(* IEC 61131-3 sources: horner-cscape-mcp/fixtures/st_programs, 6 files *)

(* ---- analog_scaling_program.st ---- *)
(* ============================================================================
 * Title:       PROGRAM AnalogScalingApp
 * Description: Multichannel Process Analog Signal Conditioner with Bounds Checking.
 * Features:
 *   - 4-Channel transmitter linear scaling to engineering units
 *   - Independent out-of-bounds detection: Wire-break and short-circuit faults
 *   - Safe value substitution during hardware transducer failure
 *   - Process alarms for high and low limit excursions
 *   - Master diagnostic health word encoding for SCADA / HMI telemetry
 * Language:    IEC 61131-3 Structured Text (Pure ST)
 * ============================================================================ *)

PROGRAM AnalogScalingApp
VAR_INPUT
    RawCh1 : REAL := 16000.0;             (* Raw ADC Channel 1: Pressure transmitter *)
    RawCh2 : REAL := 18500.0;             (* Raw ADC Channel 2: Temperature transmitter *)
    RawCh3 : REAL := 12000.0;             (* Raw ADC Channel 3: Flow rate transmitter *)
    RawCh4 : REAL := 22000.0;             (* Raw ADC Channel 4: Tank level transmitter *)
    ResetFaults : BOOL := FALSE;          (* Push button to clear sensor fault latches *)
END_VAR

VAR_OUTPUT
    Press_PSIG : REAL := 0.0;             (* Scaled pressure: 0.0 to 150.0 PSIG *)
    Temp_DegC : REAL := 0.0;              (* Scaled temperature: -20.0 to 250.0 Deg C *)
    Flow_GPM : REAL := 0.0;               (* Scaled flow rate: 0.0 to 500.0 GPM *)
    Level_Pct : REAL := 0.0;              (* Scaled vessel level: 0.0 to 100.0 % *)
    Ch1_Fault : BOOL := FALSE;            (* Channel 1 wire break or short circuit *)
    Ch2_Fault : BOOL := FALSE;            (* Channel 2 wire break or short circuit *)
    Ch3_Fault : BOOL := FALSE;            (* Channel 3 wire break or short circuit *)
    Ch4_Fault : BOOL := FALSE;            (* Channel 4 wire break or short circuit *)
    HealthStatusWord : WORD := 16#FFFF;   (* 16-bit status mask (Bit 0-3 = Channel OK) *)
    HighPressureAlarm : BOOL := FALSE;    (* Pressure above 135.0 PSIG warning *)
    HighLevelAlarm : BOOL := FALSE;       (* Level above 90.0 % overflow warning *)
END_VAR

VAR
    RawMinVal : REAL := 3200.0;           (* Raw count corresponding to 4.0 mA *)
    RawMaxVal : REAL := 32000.0;          (* Raw count corresponding to 20.0 mA *)
    BreakThreshold : REAL := 2500.0;      (* Underflow threshold declaring open circuit *)
    ShortThreshold : REAL := 32500.0;     (* Overflow threshold declaring short circuit *)
    SpanCh1 : REAL := 150.0;              (* Range span: Channel 1 *)
    SpanCh2 : REAL := 270.0;              (* Range span: Channel 2 (-20 to 250) *)
    SpanCh3 : REAL := 500.0;              (* Range span: Channel 3 *)
    SpanCh4 : REAL := 100.0;              (* Range span: Channel 4 *)
    RawSpan : REAL := 28800.0;            (* RawSpan = 32000 - 3200 *)
END_VAR

(* 1. Fault Clear *)
IF ResetFaults THEN
    Ch1_Fault := FALSE;
    Ch2_Fault := FALSE;
    Ch3_Fault := FALSE;
    Ch4_Fault := FALSE;
END_IF;

(* 2. Channel 1: Steam Header Pressure (0.0 to 150.0 PSIG) *)
IF RawCh1 < BreakThreshold OR RawCh1 > ShortThreshold THEN
    Ch1_Fault := TRUE;
    Press_PSIG := 0.0; (* Fail-safe pressure reading *)
ELSE
    Press_PSIG := ((RawCh1 - RawMinVal) / RawSpan) * SpanCh1;
    Press_PSIG := LIMIT(0.0, Press_PSIG, 150.0);
END_IF;

(* 3. Channel 2: Reactor Fluid Temperature (-20.0 to 250.0 Deg C) *)
IF RawCh2 < BreakThreshold OR RawCh2 > ShortThreshold THEN
    Ch2_Fault := TRUE;
    Temp_DegC := 25.0; (* Fail-safe ambient default *)
ELSE
    Temp_DegC := -20.0 + (((RawCh2 - RawMinVal) / RawSpan) * SpanCh2);
    Temp_DegC := LIMIT(-20.0, Temp_DegC, 250.0);
END_IF;

(* 4. Channel 3: Feed Flow Rate (0.0 to 500.0 GPM) *)
IF RawCh3 < BreakThreshold OR RawCh3 > ShortThreshold THEN
    Ch3_Fault := TRUE;
    Flow_GPM := 0.0; (* Fail-safe zero flow *)
ELSE
    Flow_GPM := ((RawCh3 - RawMinVal) / RawSpan) * SpanCh3;
    Flow_GPM := LIMIT(0.0, Flow_GPM, 500.0);
END_IF;

(* 5. Channel 4: Bulk Storage Tank Level (0.0 to 100.0 %) *)
IF RawCh4 < BreakThreshold OR RawCh4 > ShortThreshold THEN
    Ch4_Fault := TRUE;
    Level_Pct := 0.0; (* Fail-safe empty level *)
ELSE
    Level_Pct := ((RawCh4 - RawMinVal) / RawSpan) * SpanCh4;
    Level_Pct := LIMIT(0.0, Level_Pct, 100.0);
END_IF;

(* 6. Process Excursion Alarms *)
HighPressureAlarm := Press_PSIG >= 135.0 AND (NOT Ch1_Fault);
HighLevelAlarm := Level_Pct >= 90.0 AND (NOT Ch4_Fault);

(* 7. Health Status Diagnostics Word *)
IF (NOT Ch1_Fault) AND (NOT Ch2_Fault) AND (NOT Ch3_Fault) AND (NOT Ch4_Fault) THEN
    HealthStatusWord := 16#000F; (* All 4 channels healthy *)
ELSE
    HealthStatusWord := 16#0000;
END_IF;

END_PROGRAM

(* ---- batch_reactor_program.st ---- *)
(* ============================================================================
 * Title:       PROGRAM BatchReactorApp
 * Description: Automated Chemical Batch Synthesis Sequential Controller.
 * Features:
 *   - Structured sequential batch phases: Fill, Dose, Heat/Mix, Soak, Cool, Drain
 *   - Recipe parameter integration: Target volume, reagent volume, cook time
 *   - Multi-actuator control: Solvent valve, dosing pump, steam, cooling, agitator
 *   - Reactor overpressure and high-temperature emergency abort interlocks
 * Language:    IEC 61131-3 Structured Text (Pure ST)
 * ============================================================================ *)

PROGRAM BatchReactorApp
VAR_INPUT
    BatchStart : BOOL := FALSE;           (* Operator start batch recipe push button *)
    BatchAbort : BOOL := FALSE;           (* Operator emergency abort push button *)
    EStopHealthy : BOOL := TRUE;          (* Safety circuit permissive *)
    CurrentLevelPct : REAL := 0.0;        (* Vessel liquid level (0.0 to 100.0 %) *)
    CurrentTempC : REAL := 22.0;          (* Vessel liquid temperature (Deg C) *)
    VesselPressBar : REAL := 0.5;         (* Internal vessel pressure (Bar) *)
    ResetAbortPB : BOOL := FALSE;         (* Clear latched abort status *)
    TargetSolventPct : REAL := 65.0;      (* Recipe: Solvent target level (%) *)
    CookTempC : REAL := 85.0;             (* Recipe: Target reaction temperature (Deg C) *)
    CookDurationSec : REAL := 120.0;      (* Recipe: Soak hold duration at cook temperature (s) *)
    CoolTempC : REAL := 35.0;             (* Recipe: Target discharge temperature (Deg C) *)
END_VAR

VAR_OUTPUT
    SolventValve : BOOL := FALSE;         (* Feed valve: Bulk solvent *)
    ReagentPump : BOOL := FALSE;          (* Dosing pump: Catalyst / reagent *)
    AgitatorMotor : BOOL := FALSE;        (* Reaction vessel impeller agitator *)
    SteamValve : BOOL := FALSE;           (* Heating jacket steam admission valve *)
    CoolingValve : BOOL := FALSE;         (* Heating jacket chilled water admission *)
    DischargePump : BOOL := FALSE;        (* Product transfer / emptying pump *)
    BatchPhase : INT := 0;                (* Current recipe phase step code *)
    BatchComplete : BOOL := FALSE;        (* Batch cycle finished flag *)
    PressureAlarm : BOOL := FALSE;        (* Overpressure safety shutdown flag *)
    PhaseTimeSec : REAL := 0.0;           (* Elapsed duration in current phase *)
END_VAR

VAR
    ScanSec : REAL := 0.1;                (* Cyclic scan interval (seconds) *)
    DoseTimer : REAL := 0.0;              (* Reagent dosing duration timer *)
    DoseRequiredSec : REAL := 20.0;       (* Dosing run time required *)
END_VAR

(* 1. Safety Interlocks and Overpressure Protection *)
IF ResetAbortPB THEN
    PressureAlarm := FALSE;
END_IF;

IF VesselPressBar >= 3.5 THEN
    PressureAlarm := TRUE;
END_IF;

IF (NOT EStopHealthy) OR BatchAbort OR PressureAlarm THEN
    BatchPhase := 9; (* Emergency Abort *)
END_IF;

(* 2. Sequential Phase Execution *)
CASE BatchPhase OF

    0: (* PHASE_IDLE: Awaiting Recipe Start *)
        SolventValve := FALSE;
        ReagentPump := FALSE;
        AgitatorMotor := FALSE;
        SteamValve := FALSE;
        CoolingValve := FALSE;
        DischargePump := FALSE;
        PhaseTimeSec := 0.0;
        BatchComplete := FALSE;

        IF BatchStart AND EStopHealthy AND (NOT PressureAlarm) THEN
            BatchPhase := 1;
        END_IF;

    1: (* PHASE_CHARGE_SOLVENT: Fill vessel with bulk solvent *)
        SolventValve := TRUE;
        AgitatorMotor := CurrentLevelPct >= 20.0; (* Start agitator once liquid covers impeller *)
        PhaseTimeSec := PhaseTimeSec + ScanSec;

        IF CurrentLevelPct >= TargetSolventPct THEN
            SolventValve := FALSE;
            DoseTimer := 0.0;
            PhaseTimeSec := 0.0;
            BatchPhase := 2;
        END_IF;

    2: (* PHASE_DOSE_REAGENT: Meter chemical catalyst *)
        ReagentPump := TRUE;
        AgitatorMotor := TRUE;
        DoseTimer := DoseTimer + ScanSec;
        PhaseTimeSec := PhaseTimeSec + ScanSec;

        IF DoseTimer >= DoseRequiredSec THEN
            ReagentPump := FALSE;
            PhaseTimeSec := 0.0;
            BatchPhase := 3;
        END_IF;

    3: (* PHASE_HEAT: Apply steam until target cook temperature is reached *)
        AgitatorMotor := TRUE;
        SteamValve := CurrentTempC < CookTempC;
        CoolingValve := FALSE;
        PhaseTimeSec := PhaseTimeSec + ScanSec;

        IF CurrentTempC >= CookTempC THEN
            PhaseTimeSec := 0.0;
            BatchPhase := 4;
        END_IF;

    4: (* PHASE_SOAK: Hold at reaction temperature for recipe duration *)
        AgitatorMotor := TRUE;
        SteamValve := CurrentTempC < CookTempC;
        CoolingValve := CurrentTempC > (CookTempC + 2.0);
        PhaseTimeSec := PhaseTimeSec + ScanSec;

        IF PhaseTimeSec >= CookDurationSec THEN
            SteamValve := FALSE;
            PhaseTimeSec := 0.0;
            BatchPhase := 5;
        END_IF;

    5: (* PHASE_COOL: Circulate chilled water to quench reaction *)
        AgitatorMotor := TRUE;
        SteamValve := FALSE;
        CoolingValve := TRUE;
        PhaseTimeSec := PhaseTimeSec + ScanSec;

        IF CurrentTempC <= CoolTempC THEN
            CoolingValve := FALSE;
            PhaseTimeSec := 0.0;
            BatchPhase := 6;
        END_IF;

    6: (* PHASE_DISCHARGE: Transfer product out of reactor *)
        AgitatorMotor := CurrentLevelPct >= 15.0;
        DischargePump := TRUE;
        PhaseTimeSec := PhaseTimeSec + ScanSec;

        IF CurrentLevelPct <= 2.0 THEN
            DischargePump := FALSE;
            AgitatorMotor := FALSE;
            BatchComplete := TRUE;
            BatchPhase := 7;
        END_IF;

    7: (* PHASE_COMPLETE: Finished, waiting for unload acknowledge *)
        SolventValve := FALSE;
        ReagentPump := FALSE;
        AgitatorMotor := FALSE;
        SteamValve := FALSE;
        CoolingValve := FALSE;
        DischargePump := FALSE;
        BatchComplete := TRUE;

        IF NOT BatchStart THEN
            BatchPhase := 0;
        END_IF;

    9: (* PHASE_ABORT: Safe shutdown state *)
        SolventValve := FALSE;
        ReagentPump := FALSE;
        SteamValve := FALSE;
        CoolingValve := TRUE; (* Quench reactor on emergency *)
        DischargePump := FALSE;
        AgitatorMotor := FALSE;

        IF (NOT PressureAlarm) AND (NOT BatchAbort) AND EStopHealthy AND ResetAbortPB THEN
            BatchPhase := 0;
        END_IF;

    ELSE
        BatchPhase := 0;
END_CASE;

END_PROGRAM

(* ---- conveyor_sorter_program.st ---- *)
(* ============================================================================
 * Title:       PROGRAM ConveyorSorterApp
 * Description: Packaging Line Conveyor Sorter with Optical Part Classification.
 * Features:
 *   - Clean integer-based CASE finite state machine
 *   - Photoeye arrival detection and barcode/height part classification
 *   - Pneumatic diverter solenoids for Bin A, Bin B, and Reject chute
 *   - Jam detection timer with conveyor stop and visual alarm
 *   - Piece counts for total throughput and sort distribution
 * Language:    IEC 61131-3 Structured Text (Pure ST)
 * ============================================================================ *)

PROGRAM ConveyorSorterApp
VAR_INPUT
    SystemStart : BOOL := FALSE;          (* Start push button *)
    SystemStop : BOOL := FALSE;           (* Stop push button *)
    PartArrivedPE : BOOL := FALSE;        (* Optical sensor at sorting inlet *)
    PartClassCode : INT := 1;             (* Vision classifier: 1 = Bin A, 2 = Bin B, other = Reject *)
    BinA_Confirmed : BOOL := FALSE;       (* Proximity sensor confirming Bin A drop *)
    BinB_Confirmed : BOOL := FALSE;       (* Proximity sensor confirming Bin B drop *)
    RejectConfirmed : BOOL := FALSE;      (* Proximity sensor confirming Reject drop *)
    ClearFaultPB : BOOL := FALSE;         (* Fault acknowledge and reset push button *)
END_VAR

VAR_OUTPUT
    BeltMotor : BOOL := FALSE;            (* Conveyor drive motor contactor *)
    DiverterA : BOOL := FALSE;            (* Pneumatic diverter solenoid for Bin A *)
    DiverterB : BOOL := FALSE;            (* Pneumatic diverter solenoid for Bin B *)
    RejectGate : BOOL := FALSE;           (* Pneumatic reject flipper gate *)
    SystemState : INT := 0;               (* Current state machine step *)
    JamAlarm : BOOL := FALSE;             (* Parcel jam alarm indicator *)
    TotalCount : DINT := 0;               (* Total items sorted *)
    BinACount : DINT := 0;                (* Count sorted to Bin A *)
    BinBCount : DINT := 0;                (* Count sorted to Bin B *)
    RejectCount : DINT := 0;              (* Count diverted to Reject *)
END_VAR

VAR
    ScanSec : REAL := 0.1;                (* Scan period (seconds) *)
    StepTimer : REAL := 0.0;              (* Active state dwell timer *)
    JamLimitSec : REAL := 3.5;            (* Jam watchdog limit (seconds) *)
    LineRunning : BOOL := FALSE;          (* Running latch flag *)
    ActiveRoute : INT := 0;               (* Latched route for item in transit *)
END_VAR

(* 1. Safety and Start/Stop Supervisory Logic *)
IF ClearFaultPB THEN
    JamAlarm := FALSE;
END_IF;

IF SystemStop OR JamAlarm THEN
    LineRunning := FALSE;
ELSIF SystemStart AND (NOT JamAlarm) THEN
    LineRunning := TRUE;
END_IF;

(* 2. Sequential Sortation State Machine *)
CASE SystemState OF

    0: (* STATE_IDLE: Awaiting Start Command *)
        BeltMotor := FALSE;
        DiverterA := FALSE;
        DiverterB := FALSE;
        RejectGate := FALSE;
        StepTimer := 0.0;

        IF LineRunning THEN
            SystemState := 1;
        END_IF;

    1: (* STATE_WAIT_PART: Conveyor running, scanning for parts *)
        BeltMotor := TRUE;
        DiverterA := FALSE;
        DiverterB := FALSE;
        RejectGate := FALSE;

        IF NOT LineRunning THEN
            SystemState := 0;
        ELSIF PartArrivedPE THEN
            ActiveRoute := PartClassCode;
            StepTimer := 0.0;
            IF ActiveRoute = 1 THEN
                SystemState := 2; (* Route to Bin A *)
            ELSIF ActiveRoute = 2 THEN
                SystemState := 3; (* Route to Bin B *)
            ELSE
                SystemState := 4; (* Route to Reject *)
            END_IF;
        END_IF;

    2: (* STATE_DIVERT_A: Actuate Diverter A *)
        BeltMotor := TRUE;
        DiverterA := TRUE;
        StepTimer := StepTimer + ScanSec;

        IF BinA_Confirmed OR (StepTimer >= 1.5) THEN
            BinACount := BinACount + 1;
            TotalCount := TotalCount + 1;
            DiverterA := FALSE;
            SystemState := 1;
        ELSIF StepTimer >= JamLimitSec THEN
            JamAlarm := TRUE;
            SystemState := 9;
        END_IF;

    3: (* STATE_DIVERT_B: Actuate Diverter B *)
        BeltMotor := TRUE;
        DiverterB := TRUE;
        StepTimer := StepTimer + ScanSec;

        IF BinB_Confirmed OR (StepTimer >= 1.5) THEN
            BinBCount := BinBCount + 1;
            TotalCount := TotalCount + 1;
            DiverterB := FALSE;
            SystemState := 1;
        ELSIF StepTimer >= JamLimitSec THEN
            JamAlarm := TRUE;
            SystemState := 9;
        END_IF;

    4: (* STATE_REJECT: Actuate Reject Gate *)
        BeltMotor := TRUE;
        RejectGate := TRUE;
        StepTimer := StepTimer + ScanSec;

        IF RejectConfirmed OR (StepTimer >= 1.5) THEN
            RejectCount := RejectCount + 1;
            TotalCount := TotalCount + 1;
            RejectGate := FALSE;
            SystemState := 1;
        ELSIF StepTimer >= JamLimitSec THEN
            JamAlarm := TRUE;
            SystemState := 9;
        END_IF;

    9: (* STATE_JAM_FAULT: Line stopped on parcel jam *)
        BeltMotor := FALSE;
        DiverterA := FALSE;
        DiverterB := FALSE;
        RejectGate := FALSE;

        IF NOT JamAlarm THEN
            SystemState := 0;
        END_IF;

    ELSE
        SystemState := 0;
END_CASE;

END_PROGRAM

(* ---- pid_temp_control_program.st ---- *)
(* ============================================================================
 * Title:       PROGRAM PIDTemperatureApp
 * Description: Industrial Oven Closed-Loop Thermal Process Controller.
 * Features:
 *   - Raw RTD temperature input filter and scaling
 *   - Proportional-Integral-Derivative temperature loop with Anti-Windup
 *   - Time-proportional SSR heater power modulation
 *   - Forced-air cooling fan trigger on positive temperature overshoot
 *   - Hard safety latch cutting heater contactor on High-High alarm
 * Language:    IEC 61131-3 Structured Text (Pure ST)
 * ============================================================================ *)

PROGRAM PIDTemperatureApp
VAR_INPUT
    SystemEnable : BOOL := TRUE;          (* Master control loop enable *)
    TempSetpoint : REAL := 175.0;         (* Target operating temperature in Deg C *)
    RawAdcInput : REAL := 8750.0;         (* Raw ADC input counts (0 to 32000) *)
    ManualOverride : BOOL := FALSE;       (* Hand mode select *)
    ManualOutputVal : REAL := 0.0;        (* Manual output power (0.0 to 100.0 %) *)
    ResetTrip : BOOL := FALSE;            (* Over-temperature latch reset *)
END_VAR

VAR_OUTPUT
    SSR_HeaterPulse : BOOL := FALSE;      (* Solid-state relay digital pulse *)
    CoolingFanCmd : BOOL := FALSE;        (* Exhaust cooling fan contactor *)
    HeaterPowerPct : REAL := 0.0;         (* Calculated heating duty cycle (0.0 to 100.0 %) *)
    CurrentTemp : REAL := 25.0;           (* Filtered process temperature in Deg C *)
    HighTempAlarm : BOOL := FALSE;        (* Critical overtemperature trip latch *)
END_VAR

VAR
    ScanSec : REAL := 0.1;                (* Scan cycle time in seconds *)
    Kp : REAL := 3.5;                     (* Proportional gain *)
    Ki : REAL := 0.04;                    (* Integral gain (1/sec) *)
    Kd : REAL := 1.50;                    (* Derivative gain (sec) *)
    Error : REAL := 0.0;                  (* Control error (SP - PV) *)
    LastPV : REAL := 25.0;                (* Previous measurement for derivative *)
    IntegralAcc : REAL := 0.0;            (* Clamped integral accumulator *)
    RawPV : REAL := 25.0;                 (* Unfiltered converted temperature *)
    PwmAcc : REAL := 0.0;                 (* Time-proportional PWM period accumulator *)
    PwmPeriodSec : REAL := 4.0;           (* Base period for SSR cycling (seconds) *)
END_VAR

(* 1. Safety Trip Reset *)
IF ResetTrip THEN
    HighTempAlarm := FALSE;
END_IF;

(* 2. Analog Conversion: 0-32000 counts to 0.0-300.0 Deg C *)
RawPV := (RawAdcInput / 32000.0) * 300.0;

(* 1st-Order Low-Pass Filter: 20% alpha *)
CurrentTemp := (0.20 * RawPV) + (0.80 * CurrentTemp);

(* 3. High-High Safety Interlock *)
IF CurrentTemp >= 230.0 THEN
    HighTempAlarm := TRUE;
END_IF;

(* 4. Error and Closed-Loop PID Calculation *)
Error := TempSetpoint - CurrentTemp;

IF (NOT SystemEnable) OR HighTempAlarm THEN
    HeaterPowerPct := 0.0;
    IntegralAcc := 0.0;
    CoolingFanCmd := FALSE;
ELSIF ManualOverride THEN
    HeaterPowerPct := LIMIT(0.0, ManualOutputVal, 100.0);
    IntegralAcc := HeaterPowerPct;
    CoolingFanCmd := FALSE;
ELSE
    (* Anti-Reset Windup Integral Accumulation *)
    IntegralAcc := IntegralAcc + (Ki * Error * ScanSec);
    IntegralAcc := LIMIT(0.0, IntegralAcc, 100.0);

    (* PID Calculation: P + I - Derivative on Measurement *)
    HeaterPowerPct := (Kp * Error) + IntegralAcc - (Kd * (CurrentTemp - LastPV) / ScanSec);
    HeaterPowerPct := LIMIT(0.0, HeaterPowerPct, 100.0);

    (* Cooling Fan Assist on Significant Overshoot (+5.0 Deg C above SP) *)
    CoolingFanCmd := CurrentTemp >= (TempSetpoint + 5.0);
END_IF;
LastPV := CurrentTemp;

(* 5. Time-Proportional PWM SSR Trigger *)
IF HeaterPowerPct > 0.0 AND (NOT HighTempAlarm) AND SystemEnable THEN
    PwmAcc := PwmAcc + (ScanSec / PwmPeriodSec * 100.0);
    IF PwmAcc >= 100.0 THEN
        PwmAcc := 0.0;
    END_IF;
    SSR_HeaterPulse := PwmAcc < HeaterPowerPct;
ELSE
    PwmAcc := 0.0;
    SSR_HeaterPulse := FALSE;
END_IF;

END_PROGRAM

(* ---- pump_alternation_program.st ---- *)
(* ============================================================================
 * Title:       PROGRAM PumpAlternationApp
 * Description: Duplex Sump Pump Level Control with Automatic Wear Alternation.
 * Features:
 *   - Quad float switch monitoring: Stop, Lead Start, Lag Start, High Alarm
 *   - Automatic lead/lag pump duty rotation based on running hours
 *   - Pump thermal overload fault trip and automatic standby switchover
 *   - Anti-short-cycling timers protecting contactors and motor windings
 * Language:    IEC 61131-3 Structured Text (Pure ST)
 * ============================================================================ *)

PROGRAM PumpAlternationApp
VAR_INPUT
    FloatStop : BOOL := FALSE;            (* Low-level stop float (TRUE = Water above stop level) *)
    FloatLead : BOOL := FALSE;            (* Mid-level lead start float (TRUE = Start lead pump) *)
    FloatLag : BOOL := FALSE;             (* High-level lag start float (TRUE = Start lag pump) *)
    FloatHighAlarm : BOOL := FALSE;       (* Emergency wet-well overflow float *)
    Pump1_Overload : BOOL := FALSE;       (* Pump 1 motor protection trip switch *)
    Pump2_Overload : BOOL := FALSE;       (* Pump 2 motor protection trip switch *)
    AutoMode : BOOL := TRUE;              (* System automatic control mode select *)
    ResetFaults : BOOL := FALSE;          (* Fault reset push button *)
END_VAR

VAR_OUTPUT
    Pump1_Run : BOOL := FALSE;            (* Contactor digital output: Pump 1 *)
    Pump2_Run : BOOL := FALSE;            (* Contactor digital output: Pump 2 *)
    LeadPump : INT := 1;                  (* Active lead pump indicator (1 or 2) *)
    LagActive : BOOL := FALSE;            (* Secondary pump actively assisting *)
    AlarmHighLevel : BOOL := FALSE;       (* High-high overflow warning beacon *)
    Pump1_Tripped : BOOL := FALSE;        (* Pump 1 locked out on overload *)
    Pump2_Tripped : BOOL := FALSE;        (* Pump 2 locked out on overload *)
    Pump1_RunHours : REAL := 0.0;         (* Accumulated operational hours: Pump 1 *)
    Pump2_RunHours : REAL := 0.0;         (* Accumulated operational hours: Pump 2 *)
END_VAR

VAR
    ScanTimeSec : REAL := 0.1;            (* Task scan interval in seconds *)
    P1_Available : BOOL := TRUE;          (* Ready status: Pump 1 *)
    P2_Available : BOOL := TRUE;          (* Ready status: Pump 2 *)
    P1_RunTimer : REAL := 0.0;            (* Anti-short-cycle timer: Pump 1 *)
    P2_RunTimer : REAL := 0.0;            (* Anti-short-cycle timer: Pump 2 *)
    MinRunSec : REAL := 10.0;             (* Minimum run time in seconds *)
    DemandLead : BOOL := FALSE;           (* Lead pump demand latch *)
    DemandLag : BOOL := FALSE;            (* Lag pump demand latch *)
END_VAR

(* 1. Overload Fault Management *)
IF ResetFaults THEN
    Pump1_Tripped := FALSE;
    Pump2_Tripped := FALSE;
END_IF;

IF Pump1_Overload THEN
    Pump1_Tripped := TRUE;
END_IF;

IF Pump2_Overload THEN
    Pump2_Tripped := TRUE;
END_IF;

P1_Available := NOT Pump1_Tripped;
P2_Available := NOT Pump2_Tripped;
AlarmHighLevel := FloatHighAlarm;

(* 2. Level Demand Logic with Float Hysteresis *)
IF FloatLead THEN
    DemandLead := TRUE;
ELSIF NOT FloatStop THEN
    DemandLead := FALSE;
    DemandLag := FALSE;
END_IF;

IF FloatLag THEN
    DemandLag := TRUE;
END_IF;

(* 3. Lead Selection and Duty Alternation on Empty *)
IF (NOT Pump1_Run) AND (NOT Pump2_Run) THEN
    IF P1_Available AND P2_Available THEN
        IF Pump1_RunHours <= Pump2_RunHours THEN
            LeadPump := 1;
        ELSE
            LeadPump := 2;
        END_IF;
    ELSIF P1_Available THEN
        LeadPump := 1;
    ELSIF P2_Available THEN
        LeadPump := 2;
    END_IF;
ELSIF LeadPump = 1 AND (NOT P1_Available) AND P2_Available THEN
    LeadPump := 2;
ELSIF LeadPump = 2 AND (NOT P2_Available) AND P1_Available THEN
    LeadPump := 1;
END_IF;

(* 4. Pump Execution Sequencing *)
IF AutoMode THEN
    IF DemandLead THEN
        IF LeadPump = 1 THEN
            Pump1_Run := P1_Available;
            Pump2_Run := (DemandLag OR (NOT P1_Available)) AND P2_Available;
        ELSE
            Pump2_Run := P2_Available;
            Pump1_Run := (DemandLag OR (NOT P2_Available)) AND P1_Available;
        END_IF;
    ELSE
        (* Below stop level: enforce minimum runtime before shutdown *)
        IF P1_RunTimer >= MinRunSec THEN
            Pump1_Run := FALSE;
        END_IF;
        IF P2_RunTimer >= MinRunSec THEN
            Pump2_Run := FALSE;
        END_IF;
    END_IF;
ELSE
    Pump1_Run := FALSE;
    Pump2_Run := FALSE;
END_IF;

LagActive := Pump1_Run AND Pump2_Run;

(* 5. Runtime and Hour Meter Accumulation *)
IF Pump1_Run THEN
    P1_RunTimer := P1_RunTimer + ScanTimeSec;
    Pump1_RunHours := Pump1_RunHours + (ScanTimeSec / 3600.0);
ELSE
    P1_RunTimer := 0.0;
END_IF;

IF Pump2_Run THEN
    P2_RunTimer := P2_RunTimer + ScanTimeSec;
    Pump2_RunHours := Pump2_RunHours + (ScanTimeSec / 3600.0);
ELSE
    P2_RunTimer := 0.0;
END_IF;

END_PROGRAM

(* ---- traffic_control_program.st ---- *)
(* ============================================================================
 * Title:       PROGRAM TrafficControlApp
 * Description: Dual-Phase Roadway Intersection Controller with Conflict Monitoring.
 * Features:
 *   - 6-Phase state sequence: NS Green/Yellow/All-Red, EW Green/Yellow/All-Red
 *   - Vehicle inductive loop detector demand extension
 *   - Pedestrian crosswalk call buttons with Walk / Don't Walk signals
 *   - Failsafe green-conflict hardware interlock detecting conflicting greens
 *   - Emergency yellow/red flashing fault mode
 * Language:    IEC 61131-3 Structured Text (Pure ST)
 * ============================================================================ *)

PROGRAM TrafficControlApp
VAR_INPUT
    VehicleCall_NS : BOOL := FALSE;       (* Inductive loop: Vehicle waiting on North-South *)
    VehicleCall_EW : BOOL := FALSE;       (* Inductive loop: Vehicle waiting on East-West *)
    PedCall_NS : BOOL := FALSE;           (* Push button: Pedestrian crossing East-West (NS Walk) *)
    PedCall_EW : BOOL := FALSE;           (* Push button: Pedestrian crossing North-South (EW Walk) *)
    ResetConflict : BOOL := FALSE;        (* Technician key switch to reset conflict monitor *)
END_VAR

VAR_OUTPUT
    Light_NS_Red : BOOL := TRUE;          (* North-South signal: Red lamp *)
    Light_NS_Yellow : BOOL := FALSE;      (* North-South signal: Yellow lamp *)
    Light_NS_Green : BOOL := FALSE;       (* North-South signal: Green lamp *)
    Light_EW_Red : BOOL := TRUE;          (* East-West signal: Red lamp *)
    Light_EW_Yellow : BOOL := FALSE;      (* East-West signal: Yellow lamp *)
    Light_EW_Green : BOOL := FALSE;       (* East-West signal: Green lamp *)
    Ped_NS_Walk : BOOL := FALSE;          (* North-South pedestrian Walk illuminated *)
    Ped_EW_Walk : BOOL := FALSE;          (* East-West pedestrian Walk illuminated *)
    ActivePhase : INT := 1;               (* Current traffic phase step code *)
    ConflictFault : BOOL := FALSE;        (* Emergency: Conflicting greens detected *)
END_VAR

VAR
    ScanSec : REAL := 0.1;                (* Cyclic scan time (seconds) *)
    PhaseTimer : REAL := 0.0;             (* Elapsed time in active phase *)
    MinGreenSec : REAL := 10.0;           (* Minimum green interval *)
    MaxGreenSec : REAL := 30.0;           (* Maximum green interval *)
    YellowTimeSec : REAL := 3.5;          (* Yellow clearance interval *)
    AllRedTimeSec : REAL := 2.0;          (* All-red clearance safety interval *)
    PedLatched_NS : BOOL := FALSE;        (* Latched pedestrian call *)
    PedLatched_EW : BOOL := FALSE;        (* Latched pedestrian call *)
    FlashTimer : REAL := 0.0;             (* Flasher timer during conflict fault *)
    FlashState : BOOL := FALSE;           (* Flashing toggle signal *)
END_VAR

(* 1. Conflict Fault Reset and Safety Interlock *)
IF ResetConflict THEN
    ConflictFault := FALSE;
END_IF;

(* Green Conflict Monitor: Conflicting greens must never be TRUE together *)
IF Light_NS_Green AND Light_EW_Green THEN
    ConflictFault := TRUE;
END_IF;

(* 2. Latch Pedestrian Calls *)
IF PedCall_NS THEN PedLatched_NS := TRUE; END_IF;
IF PedCall_EW THEN PedLatched_EW := TRUE; END_IF;

(* 3. Conflict Fault Emergency Flashing (All Red flashing at 1 Hz) *)
IF ConflictFault THEN
    FlashTimer := FlashTimer + ScanSec;
    IF FlashTimer >= 0.5 THEN
        FlashTimer := 0.0;
        FlashState := NOT FlashState;
    END_IF;

    Light_NS_Green := FALSE;
    Light_NS_Yellow := FALSE;
    Light_NS_Red := FlashState;
    Light_EW_Green := FALSE;
    Light_EW_Yellow := FALSE;
    Light_EW_Red := FlashState;
    Ped_NS_Walk := FALSE;
    Ped_EW_Walk := FALSE;
    RETURN;
END_IF;

(* 4. Sequential Phase State Machine *)
PhaseTimer := PhaseTimer + ScanSec;

CASE ActivePhase OF

    1: (* PHASE_NS_GREEN: North-South Flowing *)
        Light_NS_Red := FALSE;
        Light_NS_Yellow := FALSE;
        Light_NS_Green := TRUE;
        Light_EW_Red := TRUE;
        Light_EW_Yellow := FALSE;
        Light_EW_Green := FALSE;
        Ped_NS_Walk := PedLatched_NS AND (PhaseTimer <= 7.0);
        Ped_EW_Walk := FALSE;

        (* Transition to NS Yellow if min green expired and opposing demand exists, or max green reached *)
        IF (PhaseTimer >= MinGreenSec AND (VehicleCall_EW OR PedLatched_EW)) OR (PhaseTimer >= MaxGreenSec) THEN
            PedLatched_NS := FALSE;
            PhaseTimer := 0.0;
            ActivePhase := 2;
        END_IF;

    2: (* PHASE_NS_YELLOW: North-South Clearance *)
        Light_NS_Green := FALSE;
        Light_NS_Yellow := TRUE;
        Light_NS_Red := FALSE;
        Light_EW_Red := TRUE;
        Ped_NS_Walk := FALSE;

        IF PhaseTimer >= YellowTimeSec THEN
            PhaseTimer := 0.0;
            ActivePhase := 3;
        END_IF;

    3: (* PHASE_ALL_RED_1: Safety Buffer before EW Green *)
        Light_NS_Yellow := FALSE;
        Light_NS_Red := TRUE;
        Light_EW_Red := TRUE;

        IF PhaseTimer >= AllRedTimeSec THEN
            PhaseTimer := 0.0;
            ActivePhase := 4;
        END_IF;

    4: (* PHASE_EW_GREEN: East-West Flowing *)
        Light_NS_Red := TRUE;
        Light_NS_Yellow := FALSE;
        Light_NS_Green := FALSE;
        Light_EW_Red := FALSE;
        Light_EW_Yellow := FALSE;
        Light_EW_Green := TRUE;
        Ped_EW_Walk := PedLatched_EW AND (PhaseTimer <= 7.0);
        Ped_NS_Walk := FALSE;

        (* Transition to EW Yellow if min green expired and opposing demand exists, or max green reached *)
        IF (PhaseTimer >= MinGreenSec AND (VehicleCall_NS OR PedLatched_NS)) OR (PhaseTimer >= MaxGreenSec) THEN
            PedLatched_EW := FALSE;
            PhaseTimer := 0.0;
            ActivePhase := 5;
        END_IF;

    5: (* PHASE_EW_YELLOW: East-West Clearance *)
        Light_EW_Green := FALSE;
        Light_EW_Yellow := TRUE;
        Light_EW_Red := FALSE;
        Light_NS_Red := TRUE;
        Ped_EW_Walk := FALSE;

        IF PhaseTimer >= YellowTimeSec THEN
            PhaseTimer := 0.0;
            ActivePhase := 6;
        END_IF;

    6: (* PHASE_ALL_RED_2: Safety Buffer before NS Green *)
        Light_EW_Yellow := FALSE;
        Light_EW_Red := TRUE;
        Light_NS_Red := TRUE;

        IF PhaseTimer >= AllRedTimeSec THEN
            PhaseTimer := 0.0;
            ActivePhase := 1;
        END_IF;

    ELSE
        ActivePhase := 1;
END_CASE;

END_PROGRAM
